// Mitsubishi GX Works2 project: b09   PLC: Q02/Q02H

PROGRAM MAIN
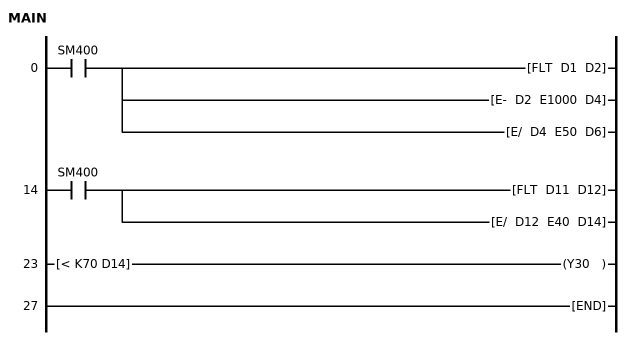
0     LD      SM400
      FLT     D1 D2
      E-      D2 E1000 D4
      E/      D4 E50 D6
14    LD      SM400
      FLT     D11 D12
      E/      D12 E40 D14
23    LD<     K70 D14
      OUT     Y30
27    END
END_PROGRAM
